{attribute 'qualified_only'}
{attribute 'strict'}
{attribute 'to_string'}
TYPE E_TCPIP_SEND_STATE :
(
	IDLE,
	CONNECT,
	SEND,
	RECEIVE,
	DISCONNECT,
	DONE,
	CONN_RESET,
	HEARTBEAT_CHECK,
	ERROR
);
END_TYPE

(* stored: Version 1.1.0.1
   DUT E_TCPIP_SEND_STATE: Id {b7d4b865-5169-4c40-b29d-668172cd65b8} *)
